% RSLogix 500 project first.RSS, saved by version 8.30.00.16 %
PROJECT "UNTITLED"    % processor: Bul.1763 MicroLogix 1100 Series B %

PROGRAM FILES
  LAD 2   7 rungs

DATA FILES
  O0 OUTPUT  4 elements
  I1 INPUT  6 elements
  S2 STATUS  66 elements
  B3 BINARY  1 elements
  T4 TIMER  1 elements
  C5 COUNTER  1 elements
  R6 CONTROL  1 elements
  N7 INTEGER  1 elements
  F8 FLOAT  1 elements

LADDER 2
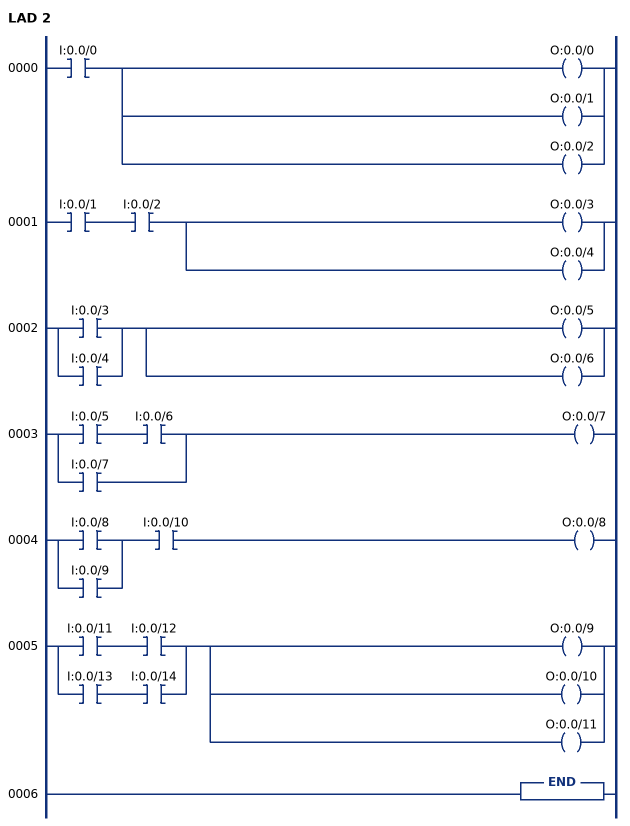
% Rung: 0 %
SOR XIC I:0.0/0 BST OTE O:0.0/0 NXB BST OTE O:0.0/1 NXB OTE O:0.0/2 BND BND EOR
% Rung: 1 %
SOR XIC I:0.0/1 XIC I:0.0/2 BST OTE O:0.0/3 NXB OTE O:0.0/4 BND EOR
% Rung: 2 %
SOR BST XIC I:0.0/3 NXB XIC I:0.0/4 BND BST OTE O:0.0/5 NXB OTE O:0.0/6 BND EOR
% Rung: 3 %
SOR BST XIC I:0.0/5 XIC I:0.0/6 NXB XIC I:0.0/7 BND OTE O:0.0/7 EOR
% Rung: 4 %
SOR BST XIC I:0.0/8 NXB XIC I:0.0/9 BND XIC I:0.0/10 OTE O:0.0/8 EOR
% Rung: 5 %
SOR BST XIC I:0.0/11 XIC I:0.0/12 NXB XIC I:0.0/13 XIC I:0.0/14 BND BST OTE O:0.0/9 NXB BST OTE O:0.0/10 NXB OTE O:0.0/11 BND BND EOR
% Rung: 6 %
SOR END EOR
